{attribute 'qualified_only'}
{attribute 'strict'}
TYPE E_OpPSBStep :
(
	START_STEP := TO_INT(E_OpStep.START_STEP)
);
END_TYPE

(* stored: Version 1.1.0.1, ProductVersion 3.1.4024.0
   DUT E_OpPSBStep: Id {3fb5b9bc-6d9e-46e9-b583-16408d8d5ba7} *)
